FUNCTION_BLOCK FB_DS
VAR_INPUT
END_VAR
VAR_OUTPUT
	{attribute 'OPC.UA.DA' := '1'}Parameter		: ST_DS_Parameter;	
	{attribute 'OPC.UA.DA' := '1'}Zustand			: ST_DS_Zustand; 
END_VAR
VAR
	Zustandscheck	: FB_DS_Zustandscheck;

	LeseDaten		: FB_DS_Input;

	IN_Status		AT %I*: USINT;
	IN_Druck		AT%I* : INT;

END_VAR

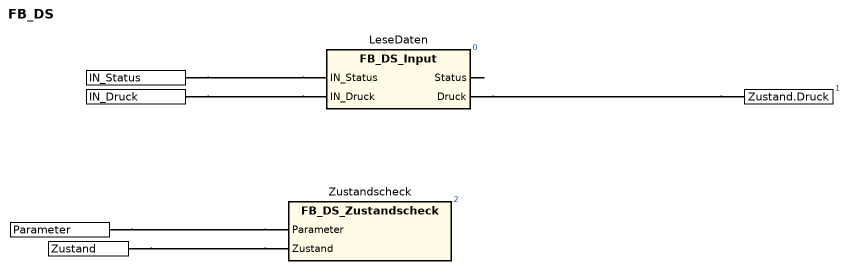
LeseDaten(IN_Status := IN_Status, IN_Druck := IN_Druck); // FB_DS_Input
Zustand.Druck := LeseDaten.Druck;
Zustandscheck(Parameter := Parameter, Zustand := Zustand); // FB_DS_Zustandscheck

END_FUNCTION_BLOCK

(* stored: Version 1.1.0.1, ProductVersion 3.1.4024.9
   POU FB_DS: Id {16265860-2a29-46f2-a014-3d873c136bb0}, SpecialFunc None *)
